(* IEC 61131-3 sources: DrakonEditor/examples/ST, 3 files *)

(* ---- IntroSFC.st ---- *)
// Autogenerated with DRAKON Editor 1.31
// IntroSFC: SFC/GRAFCET example translated to a DRAKON scan-cycle sequencer.
// Source: IntroSFC.grafcet. Call the program once per PLC scan.
// Step flags X1..X12 hold the SFC state; X1 starts active.

FUNCTION_BLOCK IntroSFC
VAR_INPUT
    I0 : BOOL;
    I1 : BOOL;
    I2 : BOOL;
    I3 : BOOL;
    I4 : BOOL;
    I5 : BOOL;
    I6 : BOOL;
    I7 : BOOL;
    I8 : BOOL;
    I9 : BOOL;
END_VAR
VAR_OUTPUT
    Q0 : BOOL;
    Q1 : BOOL;
    Q2 : BOOL;
    Q3 : BOOL;
    Q4 : BOOL;
    Q5 : BOOL;
    Q6 : BOOL;
    Q7 : BOOL;
    Q8 : BOOL;
    Q9 : BOOL;
    Q10 : BOOL;
END_VAR
VAR
    X1 : BOOL := TRUE;
    X2 : BOOL;
    X3 : BOOL;
    X4 : BOOL;
    X5 : BOOL;
    X6 : BOOL;
    X7 : BOOL;
    X8 : BOOL;
    X9 : BOOL;
    X10 : BOOL;
    X11 : BOOL;
    X12 : BOOL;
    t0 : BOOL;
    t1 : BOOL;
    t2 : BOOL;
    t3 : BOOL;
    t4 : BOOL;
    t5 : BOOL;
    t6 : BOOL;
    t7 : BOOL;
    t8 : BOOL;
    t9 : BOOL;
    t10 : BOOL;
    delayTimer : TON;
END_VAR
    // item 4
    delayTimer(IN := X12, PT := T#15S);
    // item 5
    t0 := X1 AND I0;
    t1 := X2 AND I1;
    t2 := X2 AND I2 AND NOT I1;
    t3 := X3 AND I3;
    t4 := X5 AND I4;
    t5 := X4 AND I5;
    t6 := X6 AND I6;
    t7 := X8 AND I7;
    t8 := X10 AND I8;
    t9 := X7 AND X9 AND X11 AND I9;
    t10 := X12 AND delayTimer.Q;
    // item 6
    IF t0 THEN
        // item 7
        X1 := FALSE;
        X2 := TRUE;
    ELSE
        ;
    END_IF;
    // item 10
    IF t1 THEN
        // item 11
        X2 := FALSE;
        X3 := TRUE;
    ELSE
        ;
    END_IF;
    // item 14
    IF t2 THEN
        // item 15
        X2 := FALSE;
        X5 := TRUE;
    ELSE
        ;
    END_IF;
    // item 18
    IF t3 THEN
        // item 19
        X3 := FALSE;
        X4 := TRUE;
    ELSE
        ;
    END_IF;
    // item 22
    IF t4 THEN
        // item 23
        X5 := FALSE;
        X4 := TRUE;
    ELSE
        ;
    END_IF;
    // item 26
    IF t5 THEN
        // item 27
        X4 := FALSE;
        X6 := TRUE;
        X8 := TRUE;
        X10 := TRUE;
    ELSE
        ;
    END_IF;
    // item 30
    IF t6 THEN
        // item 31
        X6 := FALSE;
        X7 := TRUE;
    ELSE
        ;
    END_IF;
    // item 34
    IF t7 THEN
        // item 35
        X8 := FALSE;
        X9 := TRUE;
    ELSE
        ;
    END_IF;
    // item 38
    IF t8 THEN
        // item 39
        X10 := FALSE;
        X11 := TRUE;
    ELSE
        ;
    END_IF;
    // item 42
    IF t9 THEN
        // item 43
        X7 := FALSE;
        X9 := FALSE;
        X11 := FALSE;
        X12 := TRUE;
    ELSE
        ;
    END_IF;
    // item 46
    IF t10 THEN
        // item 47
        X12 := FALSE;
        X1 := TRUE;
    ELSE
        ;
    END_IF;
    // item 50
    IF X10 THEN
        // item 51
        Q8 := TRUE;
    ELSE
        ;
    END_IF;
    // item 54
    IF X1 THEN
        // item 55
        Q8 := FALSE;
    ELSE
        ;
    END_IF;
    // item 58
    Q0 := X2;
    Q1 := X3;
    Q2 := X5;
    Q3 := X4;
    Q4 := X6;
    Q5 := X7;
    Q6 := X8;
    Q7 := X9;
    Q9 := X11;
    Q10 := X12;
END_FUNCTION_BLOCK

(* ---- IntroSFC_Case.st ---- *)
// Autogenerated with DRAKON Editor 1.31
// IntroSFC_Case: SFC/GRAFCET example as a DRAKON silhouette (case) machine.
// Source: IntroSFC.grafcet. Call the program once per PLC scan.
// step holds the active GRAFCET step (99 = parallel section,
// tracked by doneA/doneB/doneC).

PROGRAM IntroSFC_Case
VAR_INPUT
    I0 : BOOL;
    I1 : BOOL;
    I2 : BOOL;
    I3 : BOOL;
    I4 : BOOL;
    I5 : BOOL;
    I6 : BOOL;
    I7 : BOOL;
    I8 : BOOL;
    I9 : BOOL;
END_VAR
VAR_OUTPUT
    Q0 : BOOL;
    Q1 : BOOL;
    Q2 : BOOL;
    Q3 : BOOL;
    Q4 : BOOL;
    Q5 : BOOL;
    Q6 : BOOL;
    Q7 : BOOL;
    Q8 : BOOL;
    Q9 : BOOL;
    Q10 : BOOL;
END_VAR
VAR
    step : INT := 1;
    doneA : BOOL;
    doneB : BOOL;
    doneC : BOOL;
    delayTimer : TON;
END_VAR
    // item 5
    delayTimer(IN := (step = 12),
        PT := T#15S);
    CASE step OF
        1 :
            // item 31
            Q8 := FALSE;
            // item 32
            IF I0 THEN
                // item 33
                step := 2;
            ELSE
                ;
            END_IF;
            // item 99
            Q0 := (step = 2);
            Q1 := (step = 3);
            Q2 := (step = 5);
            Q3 := (step = 4);
            Q4 := (step = 99) AND NOT doneA;
            Q5 := (step = 99) AND doneA;
            Q6 := (step = 99) AND NOT doneB;
            Q7 := (step = 99) AND doneB;
            Q9 := (step = 99) AND doneC;
            Q10 := (step = 12);

        2 :
            // item 39
            IF I1 THEN
                // item 40
                step := 3;
            ELSE
                // item 41
                IF I2 THEN
                    // item 42
                    step := 5;
                ELSE
                    ;
                END_IF;
            END_IF;
            // item 99
            Q0 := (step = 2);
            Q1 := (step = 3);
            Q2 := (step = 5);
            Q3 := (step = 4);
            Q4 := (step = 99) AND NOT doneA;
            Q5 := (step = 99) AND doneA;
            Q6 := (step = 99) AND NOT doneB;
            Q7 := (step = 99) AND doneB;
            Q9 := (step = 99) AND doneC;
            Q10 := (step = 12);

        3 :
            // item 49
            IF I3 THEN
                // item 50
                step := 4;
            ELSE
                ;
            END_IF;
            // item 99
            Q0 := (step = 2);
            Q1 := (step = 3);
            Q2 := (step = 5);
            Q3 := (step = 4);
            Q4 := (step = 99) AND NOT doneA;
            Q5 := (step = 99) AND doneA;
            Q6 := (step = 99) AND NOT doneB;
            Q7 := (step = 99) AND doneB;
            Q9 := (step = 99) AND doneC;
            Q10 := (step = 12);

        4 :
            // item 63
            IF I5 THEN
                // item 64
                step := 99;
                doneA := FALSE;
                doneB := FALSE;
                doneC := FALSE;
            ELSE
                ;
            END_IF;
            // item 99
            Q0 := (step = 2);
            Q1 := (step = 3);
            Q2 := (step = 5);
            Q3 := (step = 4);
            Q4 := (step = 99) AND NOT doneA;
            Q5 := (step = 99) AND doneA;
            Q6 := (step = 99) AND NOT doneB;
            Q7 := (step = 99) AND doneB;
            Q9 := (step = 99) AND doneC;
            Q10 := (step = 12);

        5 :
            // item 56
            IF I4 THEN
                // item 57
                step := 4;
            ELSE
                ;
            END_IF;
            // item 99
            Q0 := (step = 2);
            Q1 := (step = 3);
            Q2 := (step = 5);
            Q3 := (step = 4);
            Q4 := (step = 99) AND NOT doneA;
            Q5 := (step = 99) AND doneA;
            Q6 := (step = 99) AND NOT doneB;
            Q7 := (step = 99) AND doneB;
            Q9 := (step = 99) AND doneC;
            Q10 := (step = 12);

        99 :
            // item 70
            IF doneA AND doneB AND doneC AND I9 THEN
                // item 71
                step := 12;
            ELSE
                ;
            END_IF;
            // item 74
            IF NOT doneC THEN
                // item 75
                Q8 := TRUE;
            ELSE
                ;
            END_IF;
            // item 78
            IF NOT doneA AND I6 THEN
                // item 79
                doneA := TRUE;
            ELSE
                ;
            END_IF;
            // item 82
            IF NOT doneB AND I7 THEN
                // item 83
                doneB := TRUE;
            ELSE
                ;
            END_IF;
            // item 86
            IF NOT doneC AND I8 THEN
                // item 87
                doneC := TRUE;
            ELSE
                ;
            END_IF;
            // item 99
            Q0 := (step = 2);
            Q1 := (step = 3);
            Q2 := (step = 5);
            Q3 := (step = 4);
            Q4 := (step = 99) AND NOT doneA;
            Q5 := (step = 99) AND doneA;
            Q6 := (step = 99) AND NOT doneB;
            Q7 := (step = 99) AND doneB;
            Q9 := (step = 99) AND doneC;
            Q10 := (step = 12);

       ELSE
            // item 93
            IF delayTimer.Q THEN
                // item 94
                step := 1;
            ELSE
                ;
            END_IF;
            // item 99
            Q0 := (step = 2);
            Q1 := (step = 3);
            Q2 := (step = 5);
            Q3 := (step = 4);
            Q4 := (step = 99) AND NOT doneA;
            Q5 := (step = 99) AND doneA;
            Q6 := (step = 99) AND NOT doneB;
            Q7 := (step = 99) AND doneB;
            Q9 := (step = 99) AND doneC;
            Q10 := (step = 12);
    END_CASE;
END_PROGRAM

(* ---- LampControl.st ---- *)
// Autogenerated with DRAKON Editor 1.31
// LampControl: minimal DRAKON Select/Case example.
// The Select icon on "mode" becomes CASE mode OF;
// the empty rightmost Case icon becomes the ELSE branch.

PROGRAM LampControl
VAR_INPUT
    mode : INT;
END_VAR
VAR_OUTPUT
    red : BOOL;
    yellow : BOOL;
    green : BOOL;
END_VAR
    CASE mode OF
        0 :
            // item 12
            red := TRUE;
            yellow := FALSE;
            green := FALSE;

        1 :
            // item 13
            red := FALSE;
            yellow := FALSE;
            green := TRUE;

       ELSE
            // item 14
            red := FALSE;
            yellow := TRUE;
            green := FALSE;
    END_CASE;
END_PROGRAM
